TYPE Range3D :
STRUCT
	X : Range;
	Y : Range;
	Z : Range;
END_STRUCT
END_TYPE

(* stored: Version 1.1.0.1
   DUT Range3D: Id {6aa17ecf-d87e-0b8c-1e23-9fee4e322b5b} *)
